TYPE AxesMultiPowerOnProcessArgs :
STRUCT
	///TRUE to power on AZI
	azi: BOOL;
	///TRUE to power on ELE
	ele: BOOL;
	///TRUE to power on ROC
	roc: BOOL;
	///TRUE to power on RON
	ron: BOOL;
	///TRUE to power on FW
	fw: BOOL;
END_STRUCT
END_TYPE

(* stored: Version 1.1.0.1, ProductVersion 3.1.4019.2
   DUT AxesMultiPowerOnProcessArgs: Id {f5d7c213-90fb-4ff5-8008-53b31a3a8d77} *)
